Fanuc KAREL source: SET_INT_REG.kl

PROGRAM T
%NOLOCKGROUP
VAR
 v0 : INTEGER
 v1 : INTEGER
 v2 : INTEGER
BEGIN
 SET_INT_REG(v0, v1, v2)
END T
